LIN {X 0,Y 14.272,Z 377.32,A -85,B 0,C 180,E1 -31509.941,E2 -31509.941} C_VEL
LIN {X 0,Y 14.475,Z 377.21,A -85,B 0,C 180,E1 -31513.8,E2 -31513.8} C_VEL
LIN {X 0,Y 23.193,Z 373.097,A -85,B 0,C 180,E1 -31515.411,E2 -31515.411} C_VEL
LIN {X 0,Y 26.111,Z 374.873,A -85,B 0,C 180,E1 -31515.647,E2 -31515.647} C_VEL
LIN {X 0,Y 26.111,Z 600,A -85,B 0,C 180,E1 -31515.647,E2 -31515.647} C_VEL
LIN {X 0,Y 26.111,Z 600,A -85,B 0,C 180,E1 -31515.647,E2 -31515.647}

QRS_NEXT_CUT()

QRS_NEXT()
QRS_HOME()

END
